(* PLC project CoDeSys External Library Template, WAGO e!COCKPIT e!COCKPIT, author 3S - Smart Software Solutions GmbH *)
(* stored: creationDateTime 2019-10-29T12:22:40.9520309, version 3.5.5.30, modificationDateTime 2019-10-24T14:40:07.960949, organization 3S - Smart Software Solutions GmbH *)
(* Library project template with all possible element types, docu and a sample project structure *)

FUNCTION fnKonwersjaHEX_STRING_TO_DEC_BYTE : BYTE
  VAR_INPUT
    sWartoscHEX : STRING(2);
  END_VAR
  VAR CONSTANT
    sTablicaReprezentacjiHEX : ARRAY[0..15] OF STRING(1) := ['0', '1', '2', '3', '4', '5', '6', '7', '8', '9', 'A', 'B', 'C', 'D', 'E', 'F'];
  END_VAR
  VAR
    sPierwszyZnak : STRING(1);
    sDrugiZnak : STRING(1);
    bPetla : BYTE;
  END_VAR

            (*			
Autor:					Paweł Kąkol, 
Prawa majątkowe: 		Solwena Sp. z o.o., 
Aktualizacje:			2018-08-24-PK - stworzenie

Opis:					Funkcja zwraca reprezentację dziesiętną jako BYTE wartości szesnastkowej podanej jako STRING;
*)

sPierwszyZnak := LEFT(sWartoscHEX, 1);
FOR bPetla := 0 TO 15 BY 1 DO
	IF sPierwszyZnak = sTablicaReprezentacjiHEX[bPetla] THEN
		fnKonwersjaHEX_STRING_TO_DEC_BYTE := bPetla * 16;
	END_IF
END_FOR
sDrugiZnak := RIGHT(sWartoscHEX, 1);
FOR bPetla := 0 TO 15 BY 1 DO
	IF sDrugiZnak = sTablicaReprezentacjiHEX[bPetla] THEN
		fnKonwersjaHEX_STRING_TO_DEC_BYTE := fnKonwersjaHEX_STRING_TO_DEC_BYTE + bPetla;
	END_IF
END_FOR

          
END_FUNCTION
